// SIMATIC S7-200 project (STEP 7-Micro/WIN), CPU 224XP REL 02.01

ORGANIZATION_BLOCK PRINCIPAL:OB1
TITLE=COMENTARIOS DEL PROGRAMA
BEGIN
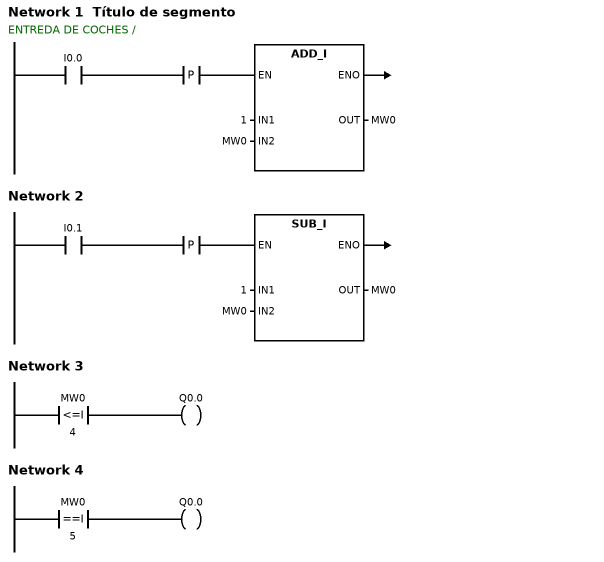
Network 1 // Título de segmento
// ENTREDA DE COCHES
// 
// (network saved uncompiled; LAD cells follow)
// row 0: c0 -| |- I0.0  c1 -|P|-  c2 [ADD_I EN:=power@row0, IN1:=1, IN2:=MW0, ENO=>power, OUT=>MW0]  c3 ->
// row 1: c2 [box]
Network 2
// (network saved uncompiled; LAD cells follow)
// row 0: c0 -| |- I0.1  c1 -|P|-  c2 [SUB_I EN:=power@row0, IN1:=1, IN2:=MW0, ENO=>power, OUT=>MW0]  c3 ->
// row 1: c2 [box]
Network 3
// (network saved uncompiled; LAD cells follow)
// row 0: c0 -|<=I|- MW0, 4  c1 -( ) Q0.0
Network 4
// (network saved uncompiled; LAD cells follow)
// row 0: c0 -|==I|- MW0, 5  c1 -( ) Q0.0
END_ORGANIZATION_BLOCK
